  #======    End of OnRobot RG Run    ======#
  # end: URCap Installation Node
  global Pallet_1_cnt_1=1
  global Pallet_1_lct=1
  global Pallet_1_lno=1
  global Pallet_1_sep= False
  global Pallet_1_tct=1
  global Pallet_2_cnt=1
  global Pallet_2_lct=1
  global Pallet_2_lno=1
  global Pallet_2_sep= False
  global Pallet_2_tct=1
  global Pallet_3_cnt=1
  global Pallet_3_lct=1
  global Pallet_3_lno=1
  global Pallet_3_sep= False
  global Pallet_3_tct=1
  global Pallet_4_cnt=1
  global Pallet_4_lct=1
  global Pallet_4_lno=1
  global Pallet_4_sep= False
  global Pallet_4_tct=1
  global Pallet_5_cnt=1
  global Pallet_5_lct=1
  global Pallet_5_lno=1
  global Pallet_5_sep= False
  global Pallet_5_tct=1
  global Pallet_6_cnt=1
  global Pallet_6_lct=1
  global Pallet_6_lno=1
  global Pallet_6_sep= False
  global Pallet_6_tct=1
  global Pallet_7_cnt=1
  global Pallet_7_lct=1
  global Pallet_7_lno=1
  global Pallet_7_sep= False
  global Pallet_7_tct=1
  global hp_p=p[.292997206297, .015070530199, .398719696079, 2.231227424716, -2.205305968938, .003332756879]
  global hp_q=[0.6887907981872559, -1.3185841006091614, -2.2963290214538574, -4.2438396416106166, -1.5708273092852991, -2.4617610613452356]
  global Approach_p=p[.299628419709, .236110783314, .306225711393, 2.247120686592, -2.190457410287, .005286769015]
  global Approach_q=[1.1426081657411131, -1.6119405231874158, -2.238066673278796, -4.008975406687, -1.5709727446182837, -2.0210788885699804]
  global ToolActionPoint_p=p[.299650785659, .236166039675, .266296927343, 2.247175696333, -2.190563516929, .005191923722]
  global ToolActionPoint_q=[1.1426595449448778, -1.669405122797066, -2.270435094833247, -3.919016023676658, -1.570828739796859, -2.0207675139058443]
  global Exit_1_p=p[.299630753541, .236110575594, .299866026681, 2.247077797521, -2.190430783414, .005165553007]
  global Exit_1_q=[1.1425796747205839, -1.6206327877446736, -2.243555545806677, -3.9948145351818125, -1.5710380713100225, -2.0210626761069825]
  global Approach_6_p=p[.473849166881, .010944546364, .326347744333, 2.247187891307, -2.190452283504, .005157127532]
  global Approach_6_q=[0.4006743431084555, -1.7402845821763329, -2.045347690582573, -4.070840021169076, -1.5685623327865725, -2.7631936708982834]
  global ToolActionPoi_6_p=p[.473861971325, .010948005681, .269628119031, 2.247173387020, -2.190520580230, .005151952022]
  global ToolActionPoi_6_q=[0.400699526071838, -1.807982584039113, -2.088192939758441, -3.9602652988829496, -1.5683959166145254, -2.762841526662024]
  global Exit_7_p=p[.473872799062, .010959164082, .320174486656, 2.247250693260, -2.190483293786, .005169534589]
  global Exit_7_q=[0.4006832242011731, -1.7471596203248332, -2.050427675247131, -4.058820625345412, -1.5685628096210884, -2.763166491184144]
  global Approach_3_p=p[.363574963744, -.129367924528, .156241055985, -2.220794216722, -2.199919030801, -.045208623402]
  global Approach_3_q=[0.11138128488887436, -1.8647028408457196, -2.3144924640643203, 2.6220084863838955, -1.5925539175727899, 0.10617900639316069]
  global ToolActionPoi_3_p=p[.363575718948, -.129360349493, .119379405887, -2.220752931187, -2.199889509891, -.045261532474]
  global ToolActionPoi_3_q=[0.11118812113991705, -1.9378115139403107, -2.3251571655273597, 2.7057444292256214, -1.593959156666843, 0.10532835870969048]
  global Exit_4_p=p[.363488717968, -.129360279908, .152553367414, -2.220605576650, -2.199818423656, -.045014129600]
  global Exit_4_q=[0.11138122528714034, -1.8718172512451403, -2.3159155845640047, 2.6303164201923104, -1.592771832142958, 0.10606686770838006]
  global Approach_4_p=p[.537418714725, .009856222325, .181969107623, 2.228346175749, 2.206374979249, -.002100509546]
  global Approach_4_q=[0.3464195728299556, -2.0103475056086353, -1.9972115755083184, 2.438913031216581, -1.5540068785309522, 0.3434899151335789]
  global ToolActionPoi_4_p=p[.537430373640, .009851549729, .143757724577, 2.228407448300, 2.206337470892, -.001995801128]
  global ToolActionPoi_4_q=[0.34624892473191754, -2.0645290813831068, -2.0089538097388058, 2.5048925119621064, -1.554978195821663, 0.3426476717013331]
  global Exit_5_p=p[.537417288040, .009861644670, .186304730584, 2.228398147696, 2.206375580336, -.002018408702]
  global Exit_5_q=[0.34643507003888757, -2.004391809501339, -1.995595932008074, 2.4313723284003093, -1.553959671648002, 0.3436143696370884]
  global Approach_5_p=p[.487656833728, .006205523921, .156383526655, 2.228227290043, 2.206418936688, -.002129849681]
  global Approach_5_q=[0.3756670057773646, -1.9883953533579586, -2.108897924422493, 2.5284854608692755, -1.5552371183989706, 0.3716393709158009]
  global ToolActionPoi_5_p=p[.487641613255, .006206234046, .116441565718, 2.228216675170, 2.206466079528, -.002174329020]
  global ToolActionPoi_5_q=[0.37552025914260817, -2.0526539287956425, -2.118428468704776, 2.602238817807578, -1.5563595930665528, 0.3707727789912685]
  global Exit_6_p=p[.487617857503, .006205113582, .155758589125, 2.228222782148, 2.206482010550, -.002251960373]
  global Exit_6_q=[0.37569323182081343, -1.9893561802299793, -2.1091504096987927, 2.52961079656755, -1.5552609602560352, 0.37162396311750623]
  global Waypoint_2_p=p[.343194716737, .015136729708, .389494181926, 2.210760885227, -2.229284741516, .003213995338]
  global Waypoint_2_q=[0.5759528279304504, -1.4386144441417237, -2.2214462757110596, -4.19599523166799, -1.5720966498004358, -2.554185930882589]
  global Waypoint_1_p=p[.343191673318, .015130816737, .281124678479, 2.210730629743, -2.229287204423, .003242849749]
  global Waypoint_1_q=[0.5764562487602234, -1.5776668987669886, -2.3315269947052, -3.9468804798521937, -1.5715869108783167, -2.5527613798724573]
  global Approach_1_p=p[.365599050903, .128716994093, .156963750112, 2.228359897720, 2.206313339354, -.001991111717]
  global Approach_1_q=[0.8015198707579335, -1.868159910238882, -2.3120160102857352, 2.608944101930586, -1.5566533247582877, 0.7967095971078699]
  global ToolActionPoi_1_p=p[.365592407714, .128732326381, .118831446023, 2.228342196091, 2.206338016038, -.001907437311]
  global ToolActionPoi_1_q=[0.8013575673110465, -1.9436775646602964, -2.3228073120119497, 2.6953040796472236, -1.5580328146535294, 0.7958391308773818]
  global Exit_2_p=p[.365569771521, .128729429257, .148672654485, 2.228270849914, 2.206438686510, -.001983247055]
  global Exit_2_q=[0.8015491366390303, -1.8841930828483378, -2.3148784637454014, 2.627844496365865, -1.556974236164315, 0.7964807748830357]
  global Approach_2_p=p[.367614890412, -.129397048939, .139517080156, -2.216595015709, -2.195337830282, -.032836288676]
  global Approach_2_q=[0.1099147796633444, -1.9054571590829283, -2.310414552688145, 2.6485091882869334, -1.5930789152725868, 0.10453771054732108]
  global ToolActionPoi_2_p=p[.367645844469, -.129390928055, .115025878284, -2.216630689520, -2.195354976828, -.032925782334]
  global ToolActionPoi_2_q=[0.10979809612066926, -1.9542862377563424, -2.3162968158722084, 2.703268213862724, -1.593967262898138, 0.10401475429578563]
  global Exit_3_p=p[.367578912567, -.129393422585, .140171166270, -2.216548159809, -2.195308788875, -.032796947710]
  global Exit_3_q=[0.10993100702720375, -1.9041553936395612, -2.310284137726036, 2.647024317379786, -1.5930822531327085, 0.10455719381548459]
  while (True):
    $ 1 "Robot Program"
    $ 2 "MoveL"
    $ 3 "hp" "breakAfter"
    movel(hp_p, a=1.2, v=0.25)
    # begin: URCap Program Node
    #   Source: OnRobot, 6.2.0, OnRobot A/S
    #   Type: RG Grip
    $ 4 "RG Grip"
on_return = rg_grip(100.0, 40.0, tool_index = 0, blocking = True, depth_comp = False, popupmsg = True)
rg_payload_set(mass = 0.0, tool_index = 0, use_guard = True)
    # end: URCap Program Node
    $ 5 "Loop 6 times"
    Loop_2 = 0
    while (Loop_2 < 6):
      $ 6 "R"
      def R_trans(pose):
      return p[pose[0], pose[1], pose[2], 0, 0, 0]
    end
    def R_rot(pose):
    return p[0, 0, 0, pose[3], pose[4], pose[5]]
  end
  def R_compute_pallet_waypoint(T_base_feature_taught, T_feature_referencePoint_taught, T_referencePoint_approach_taught, T_base_feature, T_base_referencePoint):
  local trans_referencePoint_approach_in_feature_taught = pose_sub(R_trans(pose_trans(T_feature_referencePoint_taught, T_referencePoint_approach_taught)), R_trans(T_feature_referencePoint_taught))
  local rot_referencePoint_approach_in_feature_taught = pose_trans(R_rot(T_feature_referencePoint_taught), pose_trans(R_rot(T_referencePoint_approach_taught), pose_inv(R_rot(T_feature_referencePoint_taught))))
  T_feature_referencePoint = pose_trans(pose_inv(T_base_feature), T_base_referencePoint)
  rot_referencePoint_approach = pose_trans(pose_inv(R_rot(T_feature_referencePoint)), pose_trans(rot_referencePoint_approach_in_feature_taught, R_rot(T_feature_referencePoint)))
  T_feature_approach = pose_trans(trans_referencePoint_approach_in_feature_taught, pose_trans(T_feature_referencePoint, rot_referencePoint_approach))
  T_base_approach = pose_trans(T_base_feature, T_feature_approach)
  return T_base_approach
  end
  Pallet_4_tct = 6
  if (Pallet_4_cnt > 6 or Pallet_4_cnt < 1):
    Pallet_4_cnt = 1
  end
  $ 7 "Patterns" "noBreak"
  $ 8 "Line_Pattern_5" "noBreak"
  $ 11 "Layers" "noBreak"
  if (Pallet_4_cnt < 7):
    Pallet_4_lno = 1
    Pallet_4_lct = Pallet_4_cnt
    global StartItem_5=pose_trans(p[0.0,0.0,0.0,0.0,0.0,0.0], pose_trans(p[-.000000000000, -.000000000000, -.000000000000, .000000000000, .000000000000, .000000000000], p[.297034649066, .238439755057, .270234116177, 2.210725109343, -2.229310119535, .003414031993]))
    global EndItem_5=pose_trans(p[0.0,0.0,0.0,0.0,0.0,0.0], pose_trans(p[-.000000000000, -.000000000000, -.000000000000, .000000000000, .000000000000, .000000000000], p[.171342060415, .238435045770, .270235450961, 2.210797724933, -2.229295377256, .003381978273]))
    referencePoin_3 = interpolate_pose(StartItem_5, EndItem_5, (Pallet_4_lct - 1)/5)
    direction = p[0,0,1,0,0,0]
    referencePoin_3 = pose_add (referencePoin_3,p[0.0*direction[0],0.0*direction[1],0.0*direction[2],0,0,0])
  end
  Approach_p = R_compute_pallet_waypoint(p[0.0,0.0,0.0,0.0,0.0,0.0], pose_trans(pose_inv(p[0.0,0.0,0.0,0.0,0.0,0.0]), p[0.2996507856594059,0.23616603967460775,0.2662969273431384,2.2471756963327714,-2.1905635169286577,0.0051919237216115684]), p[2.4340909054176851E-4,2.81160138336789E-5,-0.03992807672141724,-3.879481325508865E-5,1.2245647735421432E-4,-2.403664593166157E-5], p[0.0,0.0,0.0,0.0,0.0,0.0], referencePoin_3)
  Approach_p = pose_trans(p[0.2996507856594059,0.23616603967460775,0.2662969273431384,2.247175696332677,-2.190563516928566,0.005191923721586149], pose_trans(pose_inv(referencePoin_3), Approach_p))
  ToolActionPoint_p = R_compute_pallet_waypoint(p[0.0,0.0,0.0,0.0,0.0,0.0], pose_trans(pose_inv(p[0.0,0.0,0.0,0.0,0.0,0.0]), p[0.2996507856594059,0.23616603967460775,0.2662969273431384,2.2471756963327714,-2.1905635169286577,0.0051919237216115684]), p[2.7755575615628914E-17,0.0,0.0,0.0,0.0,0.0], p[0.0,0.0,0.0,0.0,0.0,0.0], referencePoin_3)
  ToolActionPoint_p = pose_trans(p[0.2996507856594059,0.23616603967460775,0.2662969273431384,2.247175696332677,-2.190563516928566,0.005191923721586149], pose_trans(pose_inv(referencePoin_3), ToolActionPoint_p))
  Exit_1_p = R_compute_pallet_waypoint(p[0.0,0.0,0.0,0.0,0.0,0.0], pose_trans(pose_inv(p[0.0,0.0,0.0,0.0,0.0,0.0]), p[0.2996507856594059,0.23616603967460775,0.2662969273431384,2.2471756963327714,-2.1905635169286577,0.0051919237216115684]), p[2.1361428246127745E-4,2.5095744851155732E-5,-0.03356846208962766,-1.2814573071368016E-4,1.0172603414222142E-4,-1.7320723826463404E-5], p[0.0,0.0,0.0,0.0,0.0,0.0], referencePoin_3)
  Exit_1_p = pose_trans(p[0.2996507856594059,0.23616603967460775,0.2662969273431384,2.247175696332677,-2.190563516928566,0.005191923721586149], pose_trans(pose_inv(referencePoin_3), Exit_1_p))
  $ 12 "At Each Item" "noBreak"
  $ 13 "Generated Movements" "noBreak"
  $ 14 "MoveJ" "noBreak"
  $ 15 "Approach" "noBreak"
  movej(get_inverse_kin(pose_trans(referencePoin_3, pose_trans(p[.227183739889, .305548767090, .267407076223, -2.247175696333, 2.190563516929, -.005191923721], Approach_p)), qnear=Approach_q), a=1.3962634015954636, v=1.0471975511965976)
  $ 16 "MoveL" "noBreak"
  $ 17 "ToolActionPoint" "noBreak"
  movel(pose_trans(referencePoin_3, pose_trans(p[.227183739889, .305548767090, .267407076223, -2.247175696333, 2.190563516929, -.005191923721], ToolActionPoint_p)), a=1.2, v=0.25)
  $ 18 "Tool action" "noBreak"
  # begin: URCap Program Node
  #   Source: OnRobot, 6.2.0, OnRobot A/S
  #   Type: RG Grip
  $ 19 "RG Grip" "noBreak"
on_return = rg_grip(73.0, 40.0, tool_index = 0, blocking = True, depth_comp = False, popupmsg = True)
rg_payload_set(mass = 0.0, tool_index = 0, use_guard = True)
  # end: URCap Program Node
  $ 20 "MoveL" "noBreak"
  $ 21 "Exit_1" "noBreak"
  movel(pose_trans(referencePoin_3, pose_trans(p[.227183739889, .305548767090, .267407076223, -2.247175696333, 2.190563516929, -.005191923721], Exit_1_p)), a=1.2, v=0.25)
  Pallet_4_sep = False
  if (Pallet_4_cnt >= 6):
    Pallet_4_cnt = 1
  else:
    Pallet_4_cnt = Pallet_4_cnt + 1
  end
  $ 22 "hp" "breakAfter"
  movel(hp_p, a=1.2, v=0.25)
  $ 23 "R2M"
  def R2M_trans(pose):
  return p[pose[0], pose[1], pose[2], 0, 0, 0]
  end
  def R2M_rot(pose):
  return p[0, 0, 0, pose[3], pose[4], pose[5]]
  end
  def R2M_compute_pallet_waypoint(T_base_feature_taught, T_feature_referencePoint_taught, T_referencePoint_approach_taught, T_base_feature, T_base_referencePoint):
  local trans_referencePoint_approach_in_feature_taught = pose_sub(R2M_trans(pose_trans(T_feature_referencePoint_taught, T_referencePoint_approach_taught)), R2M_trans(T_feature_referencePoint_taught))
  local rot_referencePoint_approach_in_feature_taught = pose_trans(R2M_rot(T_feature_referencePoint_taught), pose_trans(R2M_rot(T_referencePoint_approach_taught), pose_inv(R2M_rot(T_feature_referencePoint_taught))))
  T_feature_referencePoint = pose_trans(pose_inv(T_base_feature), T_base_referencePoint)
  rot_referencePoint_approach = pose_trans(pose_inv(R2M_rot(T_feature_referencePoint)), pose_trans(rot_referencePoint_approach_in_feature_taught, R2M_rot(T_feature_referencePoint)))
  T_feature_approach = pose_trans(trans_referencePoint_approach_in_feature_taught, pose_trans(T_feature_referencePoint, rot_referencePoint_approach))
  T_base_approach = pose_trans(T_base_feature, T_feature_approach)
  return T_base_approach
  end
  Pallet_5_tct = 6
  if (Pallet_5_cnt > 6 or Pallet_5_cnt < 1):
    Pallet_5_cnt = 1
  end
  $ 24 "Patterns" "noBreak"
  $ 25 "Line_Pattern_6" "noBreak"
  $ 28 "Line_Pattern_7" "noBreak"
  $ 31 "Layers" "noBreak"
  if (Pallet_5_cnt < 4):
    Pallet_5_lno = 1
    Pallet_5_lct = Pallet_5_cnt
    global StartItem_6=pose_trans(p[0.0,0.0,0.0,0.0,0.0,0.0], pose_trans(p[-.000000000000, -.000000000000, -.000000000000, .000000000000, .000000000000, .000000000000], p[.476303841958, .015144717273, .264840267360, 2.210749958541, -2.229240806919, .003389989203]))
    global EndItem_6=pose_trans(p[0.0,0.0,0.0,0.0,0.0,0.0], pose_trans(p[-.000000000000, -.000000000000, -.000000000000, .000000000000, .000000000000, .000000000000], p[.424584309969, .015171818780, .264878353097, 2.210828485736, -2.229320928690, .003369568903]))
    referencePoin_4 = interpolate_pose(StartItem_6, EndItem_6, (Pallet_5_lct - 1)/2)
    direction = p[0,0,1,0,0,0]
    referencePoin_4 = pose_add (referencePoin_4,p[0.0*direction[0],0.0*direction[1],0.0*direction[2],0,0,0])
  elif (Pallet_5_cnt < 7):
    Pallet_5_lno = 2
    Pallet_5_lct = Pallet_5_cnt - 3
    global StartItem_7=pose_trans(p[0.0,0.0,0.0,0.0,0.0,0.0], pose_trans(p[-.000000000000, -.000000000000, -.000000000000, .000000000000, .000000000000, .000000000000], p[.448869259714, -.010504067545, .279668869530, -3.141380868658, -.017865324447, -.004613717718]))
    global EndItem_7=pose_trans(p[0.0,0.0,0.0,0.0,0.0,0.0], pose_trans(p[-.000000000000, -.000000000000, -.000000000000, .000000000000, .000000000000, .000000000000], p[.448864663980, .041532830856, .279700594609, -3.141322233698, -.017893024746, -.004643870669]))
    referencePoin_4 = interpolate_pose(StartItem_7, EndItem_7, (Pallet_5_lct - 1)/2)
    direction = p[0,0,1,0,0,0]
    referencePoin_4 = pose_add (referencePoin_4,p[1.0E-5*direction[0],1.0E-5*direction[1],1.0E-5*direction[2],0,0,0])
  end
  Approach_6_p = R2M_compute_pallet_waypoint(p[0.0,0.0,0.0,0.0,0.0,0.0], pose_trans(pose_inv(p[0.0,0.0,0.0,0.0,0.0,0.0]), p[0.4738619713248294,0.01094800568094445,0.2696281190313883,2.247173387019771,-2.190520580229924,0.005151952022470285]), p[2.7146414670552264E-4,2.1361537813124887E-5,-0.05671897320306429,-2.427480244106472E-5,2.841312349413416E-5,-3.767624923613705E-5], p[0.0,0.0,0.0,0.0,0.0,0.0], referencePoin_4)
  Approach_6_p = pose_trans(p[0.4738619713248294,0.01094800568094445,0.2696281190313883,2.2471733870198873,-2.1905205802300376,0.005151952022511608], pose_trans(pose_inv(referencePoin_4), Approach_6_p))
  ToolActionPoi_6_p = R2M_compute_pallet_waypoint(p[0.0,0.0,0.0,0.0,0.0,0.0], pose_trans(pose_inv(p[0.0,0.0,0.0,0.0,0.0,0.0]), p[0.4738619713248294,0.01094800568094445,0.2696281190313883,2.247173387019771,-2.190520580229924,0.005151952022470285]), p[-1.734723475976807E-18,0.0,-5.551115123125783E-17,-1.348555734312709E-13,4.804316666717766E-14,-1.058681535652853E-14], p[0.0,0.0,0.0,0.0,0.0,0.0], referencePoin_4)
  ToolActionPoi_6_p = pose_trans(p[0.4738619713248294,0.01094800568094445,0.2696281190313883,2.2471733870198873,-2.1905205802300376,0.005151952022511608], pose_trans(pose_inv(referencePoin_4), ToolActionPoi_6_p))
  Exit_7_p = R2M_compute_pallet_waypoint(p[0.0,0.0,0.0,0.0,0.0,0.0], pose_trans(pose_inv(p[0.0,0.0,0.0,0.0,0.0,0.0]), p[0.4738619713248294,0.01094800568094445,0.2696281190313883,2.247173387019771,-2.190520580229924,0.005151952022470285]), p[2.2824980239933776E-4,-3.558283469817791E-6,-0.050545854539799484,2.894590649294198E-5,-1.2488270234764248E-5,-5.1338498668398555E-5], p[0.0,0.0,0.0,0.0,0.0,0.0], referencePoin_4)
  Exit_7_p = pose_trans(p[0.4738619713248294,0.01094800568094445,0.2696281190313883,2.2471733870198873,-2.1905205802300376,0.005151952022511608], pose_trans(pose_inv(referencePoin_4), Exit_7_p))
  $ 32 "At Each Item" "noBreak"
  $ 33 "Generated Movements" "noBreak"
  $ 34 "MoveJ" "noBreak"
  $ 35 "Approach_6" "noBreak"
  movej(get_inverse_kin(pose_trans(referencePoin_4, pose_trans(p[-.002428220833, .473946740727, .269690452123, -2.247173387020, 2.190520580230, -.005151952022], Approach_6_p)), qnear=Approach_6_q), a=1.3962634015954636, v=1.0471975511965976)
  $ 36 "MoveL" "noBreak"
  $ 37 "ToolActionPoi_6" "noBreak"
  movel(pose_trans(referencePoin_4, pose_trans(p[-.002428220833, .473946740727, .269690452123, -2.247173387020, 2.190520580230, -.005151952022], ToolActionPoi_6_p)), a=1.2, v=0.25)
  $ 38 "Tool action" "noBreak"
  # begin: URCap Program Node
  #   Source: OnRobot, 6.2.0, OnRobot A/S
  #   Type: RG Grip
  $ 39 "RG Grip" "noBreak"
on_return = rg_grip(100.0, 40.0, tool_index = 0, blocking = True, depth_comp = False, popupmsg = True)
rg_payload_set(mass = 0.0, tool_index = 0, use_guard = True)
  # end: URCap Program Node
  $ 40 "MoveL" "noBreak"
  $ 41 "Exit_7" "noBreak"
  movel(pose_trans(referencePoin_4, pose_trans(p[-.002428220833, .473946740727, .269690452123, -2.247173387020, 2.190520580230, -.005151952022], Exit_7_p)), a=1.2, v=0.25)
  Pallet_5_sep = False
  if (Pallet_5_cnt >= 6):
    Pallet_5_cnt = 1
  else:
    Pallet_5_cnt = Pallet_5_cnt + 1
  end
  Loop_2 = Loop_2 + 1
  end
  $ 42 "hp" "breakAfter"
  movel(hp_p, a=1.2, v=0.25)
  $ 43 "Loop 6 times"
  Loop_3 = 0
  while (Loop_3 < 6):
    $ 44 "L"
    def L_trans(pose):
    return p[pose[0], pose[1], pose[2], 0, 0, 0]
  end
  def L_rot(pose):
  return p[0, 0, 0, pose[3], pose[4], pose[5]]
  end
  def L_compute_pallet_waypoint(T_base_feature_taught, T_feature_referencePoint_taught, T_referencePoint_approach_taught, T_base_feature, T_base_referencePoint):
  local trans_referencePoint_approach_in_feature_taught = pose_sub(L_trans(pose_trans(T_feature_referencePoint_taught, T_referencePoint_approach_taught)), L_trans(T_feature_referencePoint_taught))
  local rot_referencePoint_approach_in_feature_taught = pose_trans(L_rot(T_feature_referencePoint_taught), pose_trans(L_rot(T_referencePoint_approach_taught), pose_inv(L_rot(T_feature_referencePoint_taught))))
  T_feature_referencePoint = pose_trans(pose_inv(T_base_feature), T_base_referencePoint)
  rot_referencePoint_approach = pose_trans(pose_inv(L_rot(T_feature_referencePoint)), pose_trans(rot_referencePoint_approach_in_feature_taught, L_rot(T_feature_referencePoint)))
  T_feature_approach = pose_trans(trans_referencePoint_approach_in_feature_taught, pose_trans(T_feature_referencePoint, rot_referencePoint_approach))
  T_base_approach = pose_trans(T_base_feature, T_feature_approach)
  return T_base_approach
  end
  Pallet_6_tct = 6
  if (Pallet_6_cnt > 6 or Pallet_6_cnt < 1):
    Pallet_6_cnt = 1
  end
  $ 45 "Patterns" "noBreak"
  $ 46 "Line_Pattern_8" "noBreak"
  $ 49 "Layers" "noBreak"
  if (Pallet_6_cnt < 7):
    Pallet_6_lno = 1
    Pallet_6_lct = Pallet_6_cnt
    global StartItem_8=pose_trans(p[0.0,0.0,0.0,0.0,0.0,0.0], pose_trans(p[-.000000000000, -.000000000000, -.000000000000, .000000000000, .000000000000, .000000000000], p[.299790983671, -.211736106140, .270255738881, 2.228651524880, -2.212375645079, .002577579773]))
    global EndItem_8=pose_trans(p[0.0,0.0,0.0,0.0,0.0,0.0], pose_trans(p[-.000000000000, -.000000000000, -.000000000000, .000000000000, .000000000000, .000000000000], p[.173337132643, -.211748109107, .270253593212, 2.228673183163, -2.212365101204, .002702585530]))
    referencePoin_5 = interpolate_pose(StartItem_8, EndItem_8, (Pallet_6_lct - 1)/5)
    direction = p[0,0,1,0,0,0]
    referencePoin_5 = pose_add (referencePoin_5,p[0.0*direction[0],0.0*direction[1],0.0*direction[2],0,0,0])
  end
  Approach_3_p = L_compute_pallet_waypoint(p[0.0,0.0,0.0,0.0,0.0,0.0], pose_trans(pose_inv(p[0.0,0.0,0.0,0.0,0.0,0.0]), p[0.36357571894846064,-0.129360349492781,0.11937940588682555,-2.2207529311868157,-2.1998895098905664,-0.04526153247361429]), p[0.0011491037378826702,3.4807540851411467E-4,-0.0368420915528138,-1.0986382360070954E-5,-5.911660097801395E-5,4.719051194831269E-6], p[0.0,0.0,0.0,0.0,0.0,0.0], referencePoin_5)
  Approach_3_p = pose_trans(p[0.36357571894846064,-0.129360349492781,0.11937940588682555,-2.2207529311867384,-2.19988950989049,-0.04526153247363571], pose_trans(pose_inv(referencePoin_5), Approach_3_p))
  ToolActionPoi_3_p = L_compute_pallet_waypoint(p[0.0,0.0,0.0,0.0,0.0,0.0], pose_trans(pose_inv(p[0.0,0.0,0.0,0.0,0.0,0.0]), p[0.36357571894846064,-0.129360349492781,0.11937940588682555,-2.2207529311868157,-2.1998895098905664,-0.04526153247361429]), p[0.0,0.0,0.0,-7.646747818279561E-14,-8.684025720739893E-14,-2.511364597182485E-15], p[0.0,0.0,0.0,0.0,0.0,0.0], referencePoin_5)
  ToolActionPoi_3_p = pose_trans(p[0.36357571894846064,-0.129360349492781,0.11937940588682555,-2.2207529311867384,-2.19988950989049,-0.04526153247363571], pose_trans(pose_inv(referencePoin_5), ToolActionPoi_3_p))
  Exit_4_p = L_compute_pallet_waypoint(p[0.0,0.0,0.0,0.0,0.0,0.0], pose_trans(pose_inv(p[0.0,0.0,0.0,0.0,0.0,0.0]), p[0.36357571894846064,-0.129360349492781,0.11937940588682555,-2.2207529311868157,-2.1998895098905664,-0.04526153247361429]), p[0.0010402274250875393,2.2687396069259735E-4,-0.0331569864088334,2.233173567562364E-4,1.0718108833777153E-7,-3.0534865546884656E-5], p[0.0,0.0,0.0,0.0,0.0,0.0], referencePoin_5)
  Exit_4_p = pose_trans(p[0.36357571894846064,-0.129360349492781,0.11937940588682555,-2.2207529311867384,-2.19988950989049,-0.04526153247363571], pose_trans(pose_inv(referencePoin_5), Exit_4_p))
  $ 50 "At Each Item" "noBreak"
  $ 51 "Generated Movements" "noBreak"
  $ 52 "MoveL" "noBreak"
  $ 53 "Approach_3" "noBreak"
  movel(pose_trans(referencePoin_5, pose_trans(p[.122168985295, -.365912386103, .119815319170, 2.220752931187, 2.199889509890, .045261532474], Approach_3_p)), a=1.2, v=0.25)
  $ 54 "MoveL" "noBreak"
  $ 55 "ToolActionPoi_3" "noBreak"
  movel(pose_trans(referencePoin_5, pose_trans(p[.122168985295, -.365912386103, .119815319170, 2.220752931187, 2.199889509890, .045261532474], ToolActionPoi_3_p)), a=1.2, v=0.25)
  $ 56 "Tool action" "noBreak"
  # begin: URCap Program Node
  #   Source: OnRobot, 6.2.0, OnRobot A/S
  #   Type: RG Grip
  $ 57 "RG Grip" "noBreak"
on_return = rg_grip(73.0, 40.0, tool_index = 0, blocking = True, depth_comp = False, popupmsg = True)
rg_payload_set(mass = 0.0, tool_index = 0, use_guard = True)
  # end: URCap Program Node
  $ 58 "MoveL" "noBreak"
  $ 59 "Exit_4" "noBreak"
  movel(pose_trans(referencePoin_5, pose_trans(p[.122168985295, -.365912386103, .119815319170, 2.220752931187, 2.199889509890, .045261532474], Exit_4_p)), a=1.2, v=0.25)
  Pallet_6_sep = False
  if (Pallet_6_cnt >= 6):
    Pallet_6_cnt = 1
  else:
    Pallet_6_cnt = Pallet_6_cnt + 1
  end
  $ 60 "hp" "breakAfter"
  movel(hp_p, a=1.2, v=0.25)
  $ 61 "Pallet_7"
  def Pallet_7_trans(pose):
  return p[pose[0], pose[1], pose[2], 0, 0, 0]
  end
  def Pallet_7_rot(pose):
  return p[0, 0, 0, pose[3], pose[4], pose[5]]
  end
  def Pallet_7_compute_pallet_waypoint(T_base_feature_taught, T_feature_referencePoint_taught, T_referencePoint_approach_taught, T_base_feature, T_base_referencePoint):
  local trans_referencePoint_approach_in_feature_taught = pose_sub(Pallet_7_trans(pose_trans(T_feature_referencePoint_taught, T_referencePoint_approach_taught)), Pallet_7_trans(T_feature_referencePoint_taught))
  local rot_referencePoint_approach_in_feature_taught = pose_trans(Pallet_7_rot(T_feature_referencePoint_taught), pose_trans(Pallet_7_rot(T_referencePoint_approach_taught), pose_inv(Pallet_7_rot(T_feature_referencePoint_taught))))
  T_feature_referencePoint = pose_trans(pose_inv(T_base_feature), T_base_referencePoint)
  rot_referencePoint_approach = pose_trans(pose_inv(Pallet_7_rot(T_feature_referencePoint)), pose_trans(rot_referencePoint_approach_in_feature_taught, Pallet_7_rot(T_feature_referencePoint)))
  T_feature_approach = pose_trans(trans_referencePoint_approach_in_feature_taught, pose_trans(T_feature_referencePoint, rot_referencePoint_approach))
  T_base_approach = pose_trans(T_base_feature, T_feature_approach)
  return T_base_approach
  end
  Pallet_7_tct = 6
  if (Pallet_7_cnt > 6 or Pallet_7_cnt < 1):
    Pallet_7_cnt = 1
  end
  $ 62 "Patterns" "noBreak"
  $ 63 "Line_Pattern_9" "noBreak"
  $ 66 "Line_Pattern_10" "noBreak"
  $ 69 "Layers" "noBreak"
  if (Pallet_7_cnt < 4):
    Pallet_7_lno = 1
    Pallet_7_lct = Pallet_7_cnt
    global StartItem_9=pose_trans(p[0.0,0.0,0.0,0.0,0.0,0.0], pose_trans(p[-.000000000000, -.000000000000, -.000000000000, .000000000000, .000000000000, .000000000000], p[.479682131776, .013996642884, .295411634330, 2.228576452768, -2.212472108753, .002517032241]))
    global EndItem_9=pose_trans(p[0.0,0.0,0.0,0.0,0.0,0.0], pose_trans(p[-.000000000000, -.000000000000, -.000000000000, .000000000000, .000000000000, .000000000000], p[.426950495514, .013082240255, .295389671759, 2.228677338843, -2.212180458636, .002574257636]))
    referencePoin_6 = interpolate_pose(StartItem_9, EndItem_9, (Pallet_7_lct - 1)/2)
    direction = p[0,0,1,0,0,0]
    referencePoin_6 = pose_add (referencePoin_6,p[0.0*direction[0],0.0*direction[1],0.0*direction[2],0,0,0])
  elif (Pallet_7_cnt < 7):
    Pallet_7_lno = 2
    Pallet_7_lct = Pallet_7_cnt - 3
    global StartItem_10=pose_trans(p[0.0,0.0,0.0,0.0,0.0,0.0], pose_trans(p[-.000000000000, -.000000000000, -.000000000000, .000000000000, .000000000000, .000000000000], p[.451008631659, -.015601323127, .305992329501, -3.140922848897, -.047470826142, -.003468510426]))
    global EndItem_10=pose_trans(p[0.0,0.0,0.0,0.0,0.0,0.0], pose_trans(p[-.000000000000, -.000000000000, -.000000000000, .000000000000, .000000000000, .000000000000], p[.447173071310, .041066411020, .309438872719, -3.141054589687, -.039361585224, -.003202711226]))
    referencePoin_6 = interpolate_pose(StartItem_10, EndItem_10, (Pallet_7_lct - 1)/2)
    direction = p[0,0,1,0,0,0]
    referencePoin_6 = pose_add (referencePoin_6,p[1.0E-5*direction[0],1.0E-5*direction[1],1.0E-5*direction[2],0,0,0])
  end
  Approach_4_p = Pallet_7_compute_pallet_waypoint(p[0.0,0.0,0.0,0.0,0.0,0.0], pose_trans(pose_inv(p[0.0,0.0,0.0,0.0,0.0,0.0]), p[0.5374303736396537,0.009851549729481645,0.14375772457707284,2.2284074482997447,2.206337470891794,-0.001995801128275213]), p[-1.8365180066256398E-4,1.092562219467963E-4,-0.03821078757524926,3.474196604136761E-5,-5.940870342248116E-5,-4.467402579827926E-5], p[0.0,0.0,0.0,0.0,0.0,0.0], referencePoin_6)
  Approach_4_p = pose_trans(p[0.5374303736396537,0.009851549729481645,0.14375772457707284,2.228407448299676,2.2063374708917256,-0.0019958011282429425], pose_trans(pose_inv(referencePoin_6), Approach_4_p))
  ToolActionPoi_4_p = Pallet_7_compute_pallet_waypoint(p[0.0,0.0,0.0,0.0,0.0,0.0], pose_trans(pose_inv(p[0.0,0.0,0.0,0.0,0.0,0.0]), p[0.5374303736396537,0.009851549729481645,0.14375772457707284,2.2284074482997447,2.206337470891794,-0.001995801128275213]), p[-1.734723475976807E-18,0.0,0.0,0.0,0.0,0.0], p[0.0,0.0,0.0,0.0,0.0,0.0], referencePoin_6)
  ToolActionPoi_4_p = pose_trans(p[0.5374303736396537,0.009851549729481645,0.14375772457707284,2.228407448299676,2.2063374708917256,-0.0019958011282429425], pose_trans(pose_inv(referencePoin_6), ToolActionPoi_4_p))
  Exit_5_p = Pallet_7_compute_pallet_waypoint(p[0.0,0.0,0.0,0.0,0.0,0.0], pose_trans(pose_inv(p[0.0,0.0,0.0,0.0,0.0,0.0]), p[0.5374303736396537,0.009851549729481645,0.14375772457707284,2.2284074482997447,2.206337470891794,-0.001995801128275213]), p[-1.9959886316538514E-4,1.2150042557379503E-4,-0.04254636754416796,2.4453510202692544E-5,4.019061734627443E-6,-2.1499033625642915E-5], p[0.0,0.0,0.0,0.0,0.0,0.0], referencePoin_6)
  Exit_5_p = pose_trans(p[0.5374303736396537,0.009851549729481645,0.14375772457707284,2.228407448299676,2.2063374708917256,-0.0019958011282429425], pose_trans(pose_inv(referencePoin_6), Exit_5_p))
  $ 70 "At Each Item" "noBreak"
  $ 71 "Generated Movements" "noBreak"
  $ 72 "MoveL" "noBreak"
  $ 73 "Approach_4" "noBreak"
  movel(pose_trans(referencePoin_6, pose_trans(p[-.014496021564, -.537758203614, .142129246542, -2.228407448300, -2.206337470892, .001995801128], Approach_4_p)), a=1.2, v=0.25)
  $ 74 "MoveL" "noBreak"
  $ 75 "ToolActionPoi_4" "noBreak"
  movel(pose_trans(referencePoin_6, pose_trans(p[-.014496021564, -.537758203614, .142129246542, -2.228407448300, -2.206337470892, .001995801128], ToolActionPoi_4_p)), a=1.2, v=0.25)
  $ 76 "Tool action" "noBreak"
  # begin: URCap Program Node
  #   Source: OnRobot, 6.2.0, OnRobot A/S
  #   Type: RG Grip
  $ 77 "RG Grip" "noBreak"
on_return = rg_grip(100.0, 40.0, tool_index = 0, blocking = True, depth_comp = False, popupmsg = True)
rg_payload_set(mass = 0.0, tool_index = 0, use_guard = True)
  # end: URCap Program Node
  $ 78 "MoveL" "noBreak"
  $ 79 "Exit_5" "noBreak"
  movel(pose_trans(referencePoin_6, pose_trans(p[-.014496021564, -.537758203614, .142129246542, -2.228407448300, -2.206337470892, .001995801128], Exit_5_p)), a=1.2, v=0.25)
  Pallet_7_sep = False
  if (Pallet_7_cnt >= 6):
    Pallet_7_cnt = 1
  else:
    Pallet_7_cnt = Pallet_7_cnt + 1
  end
  Loop_3 = Loop_3 + 1
  end
  $ 80 "MoveL"
  $ 81 "hp" "breakAfter"
  movel(hp_p, a=1.2, v=0.25)
  # begin: URCap Program Node
  #   Source: OnRobot, 6.2.0, OnRobot A/S
  #   Type: RG Grip
  $ 82 "RG Grip"
on_return = rg_grip(100.0, 40.0, tool_index = 0, blocking = True, depth_comp = False, popupmsg = True)
rg_payload_set(mass = 0.0, tool_index = 0, use_guard = True)
  # end: URCap Program Node
  $ 83 "Loop 12 times"
  Loop_1 = 0
  while (Loop_1 < 12):
    $ 84 "Pallet_1"
    def Pallet_1_trans(pose):
    return p[pose[0], pose[1], pose[2], 0, 0, 0]
  end
  def Pallet_1_rot(pose):
  return p[0, 0, 0, pose[3], pose[4], pose[5]]
  end
  def Pallet_1_compute_pallet_waypoint(T_base_feature_taught, T_feature_referencePoint_taught, T_referencePoint_approach_taught, T_base_feature, T_base_referencePoint):
  local trans_referencePoint_approach_in_feature_taught = pose_sub(Pallet_1_trans(pose_trans(T_feature_referencePoint_taught, T_referencePoint_approach_taught)), Pallet_1_trans(T_feature_referencePoint_taught))
  local rot_referencePoint_approach_in_feature_taught = pose_trans(Pallet_1_rot(T_feature_referencePoint_taught), pose_trans(Pallet_1_rot(T_referencePoint_approach_taught), pose_inv(Pallet_1_rot(T_feature_referencePoint_taught))))
  T_feature_referencePoint = pose_trans(pose_inv(T_base_feature), T_base_referencePoint)
  rot_referencePoint_approach = pose_trans(pose_inv(Pallet_1_rot(T_feature_referencePoint)), pose_trans(rot_referencePoint_approach_in_feature_taught, Pallet_1_rot(T_feature_referencePoint)))
  T_feature_approach = pose_trans(trans_referencePoint_approach_in_feature_taught, pose_trans(T_feature_referencePoint, rot_referencePoint_approach))
  T_base_approach = pose_trans(T_base_feature, T_feature_approach)
  return T_base_approach
  end
  Pallet_1_tct = 12
  if (Pallet_1_cnt_1 > 12 or Pallet_1_cnt_1 < 1):
    Pallet_1_cnt_1 = 1
  end
  $ 85 "Patterns" "noBreak"
  $ 86 "floor4" "noBreak"
  $ 89 "Line_Pattern_4" "noBreak"
  $ 92 "Line_Pattern_11" "noBreak"
  $ 95 "Line_Pattern_12" "noBreak"
  $ 98 "Layers" "noBreak"
  if (Pallet_1_cnt_1 < 4):
    Pallet_1_lno = 1
    Pallet_1_lct = Pallet_1_cnt_1
    global StartItem_1=pose_trans(p[0.0,0.0,0.0,0.0,0.0,0.0], pose_trans(p[-.000000000000, -.000000000000, -.000000000000, .000000000000, .000000000000, .000000000000], p[.450530530900, .038216286437, .310519820512, -3.141283005070, .024671458827, -.003216337581]))
    global EndItem_1=pose_trans(p[0.0,0.0,0.0,0.0,0.0,0.0], pose_trans(p[-.000000000000, -.000000000000, -.000000000000, .000000000000, .000000000000, .000000000000], p[.450552635246, -.010988961388, .310539318270, -3.141298717127, .024666999708, -.003239876676]))
    referencePoint = interpolate_pose(StartItem_1, EndItem_1, (Pallet_1_lct - 1)/2)
    direction = p[0,0,1,0,0,0]
    referencePoint = pose_add (referencePoint,p[3.0E-5*direction[0],3.0E-5*direction[1],3.0E-5*direction[2],0,0,0])
  elif (Pallet_1_cnt_1 < 7):
    Pallet_1_lno = 2
    Pallet_1_lct = Pallet_1_cnt_1 - 3
    global StartItem_4=pose_trans(p[0.0,0.0,0.0,0.0,0.0,0.0], pose_trans(p[-.000000000000, -.000000000000, -.000000000000, .000000000000, .000000000000, .000000000000], p[.424831985211, .013031716764, .295396183773, 2.228585492459, -2.212307486745, .002519670097]))
    global EndItem_4=pose_trans(p[0.0,0.0,0.0,0.0,0.0,0.0], pose_trans(p[-.000000000000, -.000000000000, -.000000000000, .000000000000, .000000000000, .000000000000], p[.475836865662, .014021643883, .295374286924, 2.228534269727, -2.212301690743, .002478232547]))
    referencePoint = interpolate_pose(StartItem_4, EndItem_4, (Pallet_1_lct - 1)/2)
    direction = p[0,0,1,0,0,0]
    referencePoint = pose_add (referencePoint,p[2.0E-5*direction[0],2.0E-5*direction[1],2.0E-5*direction[2],0,0,0])
  elif (Pallet_1_cnt_1 < 10):
    Pallet_1_lno = 3
    Pallet_1_lct = Pallet_1_cnt_1 - 6
    global StartItem_11=pose_trans(p[0.0,0.0,0.0,0.0,0.0,0.0], pose_trans(p[-.000000000000, -.000000000000, -.000000000000, .000000000000, .000000000000, .000000000000], p[.448848617791, -.010530165826, .279643918474, -3.141470680523, -.017863155288, -.004508053988]))
    global EndItem_11=pose_trans(p[0.0,0.0,0.0,0.0,0.0,0.0], pose_trans(p[-.000000000000, -.000000000000, -.000000000000, .000000000000, .000000000000, .000000000000], p[.448864866251, .041542775870, .279709300883, -3.141360273601, -.017931621060, -.004629582869]))
    referencePoint = interpolate_pose(StartItem_11, EndItem_11, (Pallet_1_lct - 1)/2)
    direction = p[0,0,1,0,0,0]
    referencePoint = pose_add (referencePoint,p[1.0E-5*direction[0],1.0E-5*direction[1],1.0E-5*direction[2],0,0,0])
  elif (Pallet_1_cnt_1 < 13):
    Pallet_1_lno = 4
    Pallet_1_lct = Pallet_1_cnt_1 - 9
    global StartItem_12=pose_trans(p[0.0,0.0,0.0,0.0,0.0,0.0], pose_trans(p[-.000000000000, -.000000000000, -.000000000000, .000000000000, .000000000000, .000000000000], p[.476281020793, .015161536759, .264816090095, 2.210713953344, -2.229145274570, .003345448511]))
    global EndItem_12=pose_trans(p[0.0,0.0,0.0,0.0,0.0,0.0], pose_trans(p[-.000000000000, -.000000000000, -.000000000000, .000000000000, .000000000000, .000000000000], p[.424591590215, .015165330241, .264875090798, 2.210808333375, -2.229376815489, .003330715157]))
    referencePoint = interpolate_pose(StartItem_12, EndItem_12, (Pallet_1_lct - 1)/2)
    direction = p[0,0,1,0,0,0]
    referencePoint = pose_add (referencePoint,p[0.0*direction[0],0.0*direction[1],0.0*direction[2],0,0,0])
  end
  Approach_5_p = Pallet_1_compute_pallet_waypoint(p[0.0,0.0,0.0,0.0,0.0,0.0], pose_trans(pose_inv(p[0.0,0.0,0.0,0.0,0.0,0.0]), p[0.48764161325454886,0.006206234045797706,0.11644156571844112,2.228216675170024,2.206466079527706,-0.0021743290203899914]), p[-2.0179704340587794E-4,1.3972700138448202E-4,-0.039941209670827094,-3.811933175183371E-5,2.054607624485041E-6,2.6227797710732764E-5], p[0.0,0.0,0.0,0.0,0.0,0.0], referencePoint)
  Approach_5_p = pose_trans(p[0.48764161325454886,0.006206234045797706,0.11644156571844112,2.2282166751700236,2.206466079527706,-0.0021743290203649237], pose_trans(pose_inv(referencePoint), Approach_5_p))
  ToolActionPoi_5_p = Pallet_1_compute_pallet_waypoint(p[0.0,0.0,0.0,0.0,0.0,0.0], pose_trans(pose_inv(p[0.0,0.0,0.0,0.0,0.0,0.0]), p[0.48764161325454886,0.006206234045797706,0.11644156571844112,2.228216675170024,2.206466079527706,-0.0021743290203899914]), p[0.0,0.0,0.0,1.3917686447761917E-14,1.3713856439334642E-14,9.213007960695569E-17], p[0.0,0.0,0.0,0.0,0.0,0.0], referencePoint)
  ToolActionPoi_5_p = pose_trans(p[0.48764161325454886,0.006206234045797706,0.11644156571844112,2.2282166751700236,2.206466079527706,-0.0021743290203649237], pose_trans(pose_inv(referencePoint), ToolActionPoi_5_p))
  Exit_6_p = Pallet_1_compute_pallet_waypoint(p[0.0,0.0,0.0,0.0,0.0,0.0], pose_trans(pose_inv(p[0.0,0.0,0.0,0.0,0.0,0.0]), p[0.48764161325454886,0.006206234045797706,0.11644156571844112,2.228216675170024,2.206466079527706,-0.0021743290203899914]), p[-1.9944140674679582E-4,9.880890937075115E-5,-0.03931640058660771,4.590928331983132E-5,-2.419032902647042E-5,-4.632521359925457E-6], p[0.0,0.0,0.0,0.0,0.0,0.0], referencePoint)
  Exit_6_p = pose_trans(p[0.48764161325454886,0.006206234045797706,0.11644156571844112,2.2282166751700236,2.206466079527706,-0.0021743290203649237], pose_trans(pose_inv(referencePoint), Exit_6_p))
  $ 99 "At Each Item" "noBreak"
  $ 100 "Generated Movements" "noBreak"
  $ 101 "MoveL" "noBreak"
  $ 102 "Approach_5" "noBreak"
  movel(pose_trans(referencePoint, pose_trans(p[-.010406280350, -.487917945150, .114975156776, -2.228216675170, -2.206466079528, .002174329020], Approach_5_p)), a=1.2, v=0.25)
  $ 103 "MoveL" "noBreak"
  $ 104 "ToolActionPoi_5" "noBreak"
  movel(pose_trans(referencePoint, pose_trans(p[-.010406280350, -.487917945150, .114975156776, -2.228216675170, -2.206466079528, .002174329020], ToolActionPoi_5_p)), a=1.2, v=0.25)
  $ 105 "Tool action" "noBreak"
  # begin: URCap Program Node
  #   Source: OnRobot, 6.2.0, OnRobot A/S
  #   Type: RG Grip
  $ 106 "RG Grip" "noBreak"
on_return = rg_grip(73.0, 40.0, tool_index = 0, blocking = True, depth_comp = False, popupmsg = True)
rg_payload_set(mass = 0.0, tool_index = 0, use_guard = True)
  # end: URCap Program Node
  $ 107 "MoveL" "noBreak"
  $ 108 "Exit_6" "noBreak"
  movel(pose_trans(referencePoint, pose_trans(p[-.010406280350, -.487917945150, .114975156776, -2.228216675170, -2.206466079528, .002174329020], Exit_6_p)), a=1.2, v=0.25)
  Pallet_1_sep = False
  if (Pallet_1_cnt_1 >= 12):
    Pallet_1_cnt_1 = 1
  else:
    Pallet_1_cnt_1 = Pallet_1_cnt_1 + 1
  end
  $ 109 "MoveL"
  $ 110 "Waypoint_2" "breakAfter"
  movel(Waypoint_2_p, a=1.2, v=0.25)
  $ 111 "Waypoint_1" "breakAfter"
  movel(Waypoint_1_p, a=1.2, v=0.25)
  $ 112 "Wait: 1.0"
  sleep(1.0)
  $ 113 "If analog_in[0]<5"
  if (get_standard_analog_in(0)<5):
    $ 114 "MoveL"
    $ 115 "hp" "breakAfter"
    movel(hp_p, a=1.2, v=0.25)
    $ 116 "Pallet_2"
    def Pallet_2_trans(pose):
    return p[pose[0], pose[1], pose[2], 0, 0, 0]
  end
  def Pallet_2_rot(pose):
  return p[0, 0, 0, pose[3], pose[4], pose[5]]
  end
  def Pallet_2_compute_pallet_waypoint(T_base_feature_taught, T_feature_referencePoint_taught, T_referencePoint_approach_taught, T_base_feature, T_base_referencePoint):
  local trans_referencePoint_approach_in_feature_taught = pose_sub(Pallet_2_trans(pose_trans(T_feature_referencePoint_taught, T_referencePoint_approach_taught)), Pallet_2_trans(T_feature_referencePoint_taught))
  local rot_referencePoint_approach_in_feature_taught = pose_trans(Pallet_2_rot(T_feature_referencePoint_taught), pose_trans(Pallet_2_rot(T_referencePoint_approach_taught), pose_inv(Pallet_2_rot(T_feature_referencePoint_taught))))
  T_feature_referencePoint = pose_trans(pose_inv(T_base_feature), T_base_referencePoint)
  rot_referencePoint_approach = pose_trans(pose_inv(Pallet_2_rot(T_feature_referencePoint)), pose_trans(rot_referencePoint_approach_in_feature_taught, Pallet_2_rot(T_feature_referencePoint)))
  T_feature_approach = pose_trans(trans_referencePoint_approach_in_feature_taught, pose_trans(T_feature_referencePoint, rot_referencePoint_approach))
  T_base_approach = pose_trans(T_base_feature, T_feature_approach)
  return T_base_approach
  end
  Pallet_2_tct = 6
  if (Pallet_2_cnt > 6 or Pallet_2_cnt < 1):
    Pallet_2_cnt = 1
  end
  $ 117 "Patterns" "noBreak"
  $ 118 "Line_Pattern_2" "noBreak"
  $ 121 "Layers" "noBreak"
  if (Pallet_2_cnt < 7):
    Pallet_2_lno = 1
    Pallet_2_lct = Pallet_2_cnt
    global StartItem_2=pose_trans(p[0.0,0.0,0.0,0.0,0.0,0.0], pose_trans(p[-.000000000000, -.000000000000, -.000000000000, .000000000000, .000000000000, .000000000000], p[.171332582266, .238438039663, .270227808924, 2.210831836834, -2.229181398064, .003379452431]))
    global EndItem_2=pose_trans(p[0.0,0.0,0.0,0.0,0.0,0.0], pose_trans(p[-.000000000000, -.000000000000, -.000000000000, .000000000000, .000000000000, .000000000000], p[.297031796720, .238465538917, .270258817449, 2.210814066008, -2.229326692589, .003334431080]))
    referencePoin_1 = interpolate_pose(StartItem_2, EndItem_2, (Pallet_2_lct - 1)/5)
    direction = p[0,0,1,0,0,0]
    referencePoin_1 = pose_add (referencePoin_1,p[0.0*direction[0],0.0*direction[1],0.0*direction[2],0,0,0])
  end
  Approach_1_p = Pallet_2_compute_pallet_waypoint(p[0.0,0.0,0.0,0.0,0.0,0.0], pose_trans(pose_inv(p[0.0,0.0,0.0,0.0,0.0,0.0]), p[0.3655924077144329,0.12873232638075274,0.11883144602328854,2.228342196091278,2.2063380160380115,-0.00190743731132561]), p[-2.0279424699348736E-4,1.3026179581931974E-4,-0.038131546004486774,3.423419512379672E-5,-4.128359992895348E-5,1.8976378753760003E-5], p[0.0,0.0,0.0,0.0,0.0,0.0], referencePoin_1)
  Approach_1_p = pose_trans(p[0.3655924077144329,0.12873232638075274,0.11883144602328854,2.2283421960912784,2.206338016038011,-0.001907437311333347], pose_trans(pose_inv(referencePoin_1), Approach_1_p))
  ToolActionPoi_1_p = Pallet_2_compute_pallet_waypoint(p[0.0,0.0,0.0,0.0,0.0,0.0], pose_trans(pose_inv(p[0.0,0.0,0.0,0.0,0.0,0.0]), p[0.3655924077144329,0.12873232638075274,0.11883144602328854,2.228342196091278,2.2063380160380115,-0.00190743731132561]), p[0.0,0.0,0.0,-6.857990737796355E-14,1.3716458524548604E-14,-3.201471138430769E-15], p[0.0,0.0,0.0,0.0,0.0,0.0], referencePoin_1)
  ToolActionPoi_1_p = pose_trans(p[0.3655924077144329,0.12873232638075274,0.11883144602328854,2.2283421960912784,2.206338016038011,-0.001907437311333347], pose_trans(pose_inv(referencePoin_1), ToolActionPoi_1_p))
  Exit_2_p = Pallet_2_compute_pallet_waypoint(p[0.0,0.0,0.0,0.0,0.0,0.0], pose_trans(pose_inv(p[0.0,0.0,0.0,0.0,0.0,0.0]), p[0.3655924077144329,0.12873232638075274,0.11883144602328854,2.228342196091278,2.2063380160380115,-0.00190743731132561]), p[-1.4987628035748046E-4,7.401532569101255E-5,-0.029840749019581322,4.8162793645755666E-5,-2.0027444047447927E-5,-7.779199247090566E-5], p[0.0,0.0,0.0,0.0,0.0,0.0], referencePoin_1)
  Exit_2_p = pose_trans(p[0.3655924077144329,0.12873232638075274,0.11883144602328854,2.2283421960912784,2.206338016038011,-0.001907437311333347], pose_trans(pose_inv(referencePoin_1), Exit_2_p))
  $ 122 "At Each Item" "noBreak"
  $ 123 "Generated Movements" "noBreak"
  $ 124 "MoveL" "noBreak"
  $ 125 "Approach_1" "noBreak"
  movel(pose_trans(referencePoin_1, pose_trans(p[-.131770826506, -.364680842518, .118300741249, -2.228342196091, -2.206338016038, .001907437311], Approach_1_p)), a=1.2, v=0.25)
  $ 126 "MoveL" "noBreak"
  $ 127 "ToolActionPoi_1" "noBreak"
  movel(pose_trans(referencePoin_1, pose_trans(p[-.131770826506, -.364680842518, .118300741249, -2.228342196091, -2.206338016038, .001907437311], ToolActionPoi_1_p)), a=1.2, v=0.25)
  $ 128 "Tool action" "noBreak"
  # begin: URCap Program Node
  #   Source: OnRobot, 6.2.0, OnRobot A/S
  #   Type: RG Grip
  $ 129 "RG Grip" "noBreak"
on_return = rg_grip(100.0, 40.0, tool_index = 0, blocking = True, depth_comp = False, popupmsg = True)
rg_payload_set(mass = 0.0, tool_index = 0, use_guard = True)
  # end: URCap Program Node
  $ 130 "MoveL" "noBreak"
  $ 131 "Exit_2" "noBreak"
  movel(pose_trans(referencePoin_1, pose_trans(p[-.131770826506, -.364680842518, .118300741249, -2.228342196091, -2.206338016038, .001907437311], Exit_2_p)), a=1.2, v=0.25)
  Pallet_2_sep = False
  if (Pallet_2_cnt >= 6):
    Pallet_2_cnt = 1
  else:
    Pallet_2_cnt = Pallet_2_cnt + 1
  end
  else:
    $ 132 "Else" "noBreak"
    $ 133 "MoveL"
    $ 134 "hp" "breakAfter"
    movel(hp_p, a=1.2, v=0.25)
    $ 135 "Pallet_3"
    def Pallet_3_trans(pose):
    return p[pose[0], pose[1], pose[2], 0, 0, 0]
  end
  def Pallet_3_rot(pose):
  return p[0, 0, 0, pose[3], pose[4], pose[5]]
  end
  def Pallet_3_compute_pallet_waypoint(T_base_feature_taught, T_feature_referencePoint_taught, T_referencePoint_approach_taught, T_base_feature, T_base_referencePoint):
  local trans_referencePoint_approach_in_feature_taught = pose_sub(Pallet_3_trans(pose_trans(T_feature_referencePoint_taught, T_referencePoint_approach_taught)), Pallet_3_trans(T_feature_referencePoint_taught))
  local rot_referencePoint_approach_in_feature_taught = pose_trans(Pallet_3_rot(T_feature_referencePoint_taught), pose_trans(Pallet_3_rot(T_referencePoint_approach_taught), pose_inv(Pallet_3_rot(T_feature_referencePoint_taught))))
  T_feature_referencePoint = pose_trans(pose_inv(T_base_feature), T_base_referencePoint)
  rot_referencePoint_approach = pose_trans(pose_inv(Pallet_3_rot(T_feature_referencePoint)), pose_trans(rot_referencePoint_approach_in_feature_taught, Pallet_3_rot(T_feature_referencePoint)))
  T_feature_approach = pose_trans(trans_referencePoint_approach_in_feature_taught, pose_trans(T_feature_referencePoint, rot_referencePoint_approach))
  T_base_approach = pose_trans(T_base_feature, T_feature_approach)
  return T_base_approach
  end
  Pallet_3_tct = 6
  if (Pallet_3_cnt > 6 or Pallet_3_cnt < 1):
    Pallet_3_cnt = 1
  end
  $ 136 "Patterns" "noBreak"
  $ 137 "Line_Pattern_3" "noBreak"
  $ 140 "Layers" "noBreak"
  if (Pallet_3_cnt < 7):
    Pallet_3_lno = 1
    Pallet_3_lct = Pallet_3_cnt
    global StartItem_3=pose_trans(p[0.0,0.0,0.0,0.0,0.0,0.0], pose_trans(p[-.000000000000, -.000000000000, -.000000000000, .000000000000, .000000000000, .000000000000], p[.173324016410, -.211754342694, .270267675435, 2.228638551560, -2.212441755069, .002769422738]))
    global EndItem_3=pose_trans(p[0.0,0.0,0.0,0.0,0.0,0.0], pose_trans(p[-.000000000000, -.000000000000, -.000000000000, .000000000000, .000000000000, .000000000000], p[.299778781186, -.211741973517, .270237077971, 2.228649089429, -2.212310869989, .002462638281]))
    referencePoin_2 = interpolate_pose(StartItem_3, EndItem_3, (Pallet_3_lct - 1)/5)
    direction = p[0,0,1,0,0,0]
    referencePoin_2 = pose_add (referencePoin_2,p[0.0*direction[0],0.0*direction[1],0.0*direction[2],0,0,0])
  end
  Approach_2_p = Pallet_3_compute_pallet_waypoint(p[0.0,0.0,0.0,0.0,0.0,0.0], pose_trans(pose_inv(p[0.0,0.0,0.0,0.0,0.0,0.0]), p[0.3676458444694583,-0.1293909280545595,0.11502587828448332,-2.216630689520228,-2.195354976827886,-0.0329257823341622]), p[7.336573816587866E-4,-4.367277287747884E-5,-0.024480192080145693,6.755448687663425E-5,-1.359384381890015E-5,-7.2585901317533225E-6], p[0.0,0.0,0.0,0.0,0.0,0.0], referencePoin_2)
  Approach_2_p = pose_trans(p[0.3676458444694583,-0.1293909280545595,0.11502587828448332,-2.216630689520228,-2.195354976827886,-0.03292578233415494], pose_trans(pose_inv(referencePoin_2), Approach_2_p))
  ToolActionPoi_2_p = Pallet_3_compute_pallet_waypoint(p[0.0,0.0,0.0,0.0,0.0,0.0], pose_trans(pose_inv(p[0.0,0.0,0.0,0.0,0.0,0.0]), p[0.3676458444694583,-0.1293909280545595,0.11502587828448332,-2.216630689520228,-2.195354976827886,-0.0329257823341622]), p[-2.7755575615628914E-17,0.0,0.0,0.0,0.0,0.0], p[0.0,0.0,0.0,0.0,0.0,0.0], referencePoin_2)
  ToolActionPoi_2_p = pose_trans(p[0.3676458444694583,-0.1293909280545595,0.11502587828448332,-2.216630689520228,-2.195354976827886,-0.03292578233415494], pose_trans(pose_inv(referencePoin_2), ToolActionPoi_2_p))
  Exit_3_p = Pallet_3_compute_pallet_waypoint(p[0.0,0.0,0.0,0.0,0.0,0.0], pose_trans(pose_inv(p[0.0,0.0,0.0,0.0,0.0,0.0]), p[0.3676458444694583,-0.1293909280545595,0.11502587828448332,-2.216630689520228,-2.195354976827886,-0.0329257823341622]), p[7.566999438936434E-4,-8.002517894445393E-5,-0.02513386152427892,1.2362428960152833E-4,6.838394605361467E-6,-1.4326348575695179E-5], p[0.0,0.0,0.0,0.0,0.0,0.0], referencePoin_2)
  Exit_3_p = pose_trans(p[0.3676458444694583,-0.1293909280545595,0.11502587828448332,-2.216630689520228,-2.195354976827886,-0.03292578233415494], pose_trans(pose_inv(referencePoin_2), Exit_3_p))
  $ 141 "At Each Item" "noBreak"
  $ 142 "Generated Movements" "noBreak"
  $ 143 "MoveL" "noBreak"
  $ 144 "Approach_2" "noBreak"
  movel(pose_trans(referencePoin_2, pose_trans(p[.122303008962, -.368815567665, .118968411524, 2.216630689520, 2.195354976828, .032925782334], Approach_2_p)), a=1.2, v=0.25)
  $ 145 "MoveL" "noBreak"
  $ 146 "ToolActionPoi_2" "noBreak"
  movel(pose_trans(referencePoin_2, pose_trans(p[.122303008962, -.368815567665, .118968411524, 2.216630689520, 2.195354976828, .032925782334], ToolActionPoi_2_p)), a=1.2, v=0.25)
  $ 147 "Tool action" "noBreak"
  # begin: URCap Program Node
  #   Source: OnRobot, 6.2.0, OnRobot A/S
  #   Type: RG Grip
  $ 148 "RG Grip" "noBreak"
on_return = rg_grip(100.0, 40.0, tool_index = 0, blocking = True, depth_comp = False, popupmsg = True)
rg_payload_set(mass = 0.0, tool_index = 0, use_guard = True)
  # end: URCap Program Node
  $ 149 "MoveL" "noBreak"
  $ 150 "Exit_3" "noBreak"
  movel(pose_trans(referencePoin_2, pose_trans(p[.122303008962, -.368815567665, .118968411524, 2.216630689520, 2.195354976828, .032925782334], Exit_3_p)), a=1.2, v=0.25)
  Pallet_3_sep = False
  if (Pallet_3_cnt >= 6):
    Pallet_3_cnt = 1
  else:
    Pallet_3_cnt = Pallet_3_cnt + 1
  end
  end
  Loop_1 = Loop_1 + 1
  end
  $ 151 "hp" "breakAfter"
  movel(hp_p, a=1.2, v=0.25)
  $ 152 "Halt"
  halt
  end
end
